FUNCTION_BLOCK FB_Evt_EventClasses EXTENDS FB_BA_View
VAR
	{region 'Standard'}
		// Intention:				Demonstration of a standard use-case:
		//							- Declaration of event classes for desired event-types and alarm-modes.
		//							  (See "FB_BA_EC01" for complete example of this standard use-case).
		//							- Applies event behaviour that just works.
		EC_Std01					: FB_BA_EC := (
										iParent							:= THIS^,
										nInstanceID						:= 200,
										sDescription					:= '{Standard EC (Extended Alarm)}',
										eEventType						:= E_BA_EventType.eAlarm,
										eAlarmMode						:= E_BA_AlarmMode.eExtended
									);
		EC_Std02					: FB_BA_EC := (
										iParent							:= THIS^,
										nInstanceID						:= 201,
										sDescription					:= '{Standard EC (Standard Alarm)}',
										eEventType						:= E_BA_EventType.eAlarm,
										eAlarmMode						:= E_BA_AlarmMode.eStandard
									);
		EC_Std03					: FB_BA_EC := (
										iParent							:= THIS^,
										nInstanceID						:= 202,
										sDescription					:= '{Standard EC (Simple Alarm)}',
										eEventType						:= E_BA_EventType.eAlarm,
										eAlarmMode						:= E_BA_AlarmMode.eSimple
									);

		// Intention:				Assignment of an object's event class reference.
		SimpleAlm01					: FB_BA_BI := (
										iParent							:= THIS^,
										sDescription					:= '{Some simple alarm}',
										nEventClassID					:= 202,
										sInactiveText					:= 'Normal',
										sActiveText						:= 'Alarm'
									);
	{endregion}
	{region 'Customize default settings'}
		// Intention:				Demonstration of customizing events default behaviour by settings modification:
		//							- No difference in code to "standard use-case".
		//							  (Use implementation of the same event classes)
		//							- The following parameters are editable per alarm-mode (See "BA_Param"):
		//							  - Acknowledge Flags
		//							  - Event Enable Flags
		
		// Sample:					How to adjust the default-settings of event-classes?
		//							- No acknowledgement should be required for any "simple" events.
		//							  BA_Param.aAckFlags_Simple := [ FALSE, FALSE, FALSE ];
	{endregion}
	{region 'Individual parameters'}
		// Intention:				Demonstration of customizing individual event-classes and objects:
		// 							- Initialization of an event-classes "AcknowledgeRequired" flags.
		EC_Cstm01					: FB_BA_EC := (
										iParent							:= THIS^,
										nInstanceID						:= 220,
										sDescription					:= '{Customized EC (Alarm 1)}',
										eEventType						:= E_BA_EventType.eAlarm,
										aAcknowledgeRequired			:= [ TRUE, TRUE, TRUE ]
									);
		EC_Cstm02					: FB_BA_EC := (
										iParent							:= THIS^,
										nInstanceID						:= 221,
										sDescription					:= '{Customized EC (Alarm 2)}',
										eEventType						:= E_BA_EventType.eAlarm,
										aAcknowledgeRequired			:= [ TRUE, FALSE, FALSE ]
									);
		EC_Cstm03					: FB_BA_EC := (
										iParent							:= THIS^,
										nInstanceID						:= 222,
										sDescription					:= '{Customized EC (Alarm 3)}',
										eEventType						:= E_BA_EventType.eAlarm,
										aAcknowledgeRequired			:= [ FALSE, FALSE, FALSE ]
									);
										 
		// Sample:					How to initialize individual objects?
		// Intention:				- Assignment of an object's event class reference.
		// 							- Initialization of an object's "EventEnable" flags.
		Alm01						: FB_BA_BI := (
										iParent							:= THIS^,
										sDescription					:= '{Some alarm without acknowledgement}',
										nEventClassID					:= 222,
										aEventEnable					:= [ TRUE, TRUE, TRUE ],
										sInactiveText					:= 'Normal',
										sActiveText						:= 'Alarm'
									);
		Alm02						: FB_BA_BI := (
										iParent							:= THIS^,
										sDescription					:= '{Some alarm with acknowledgement}',
										nEventClassID					:= 220,
										aEventEnable					:= [ TRUE, TRUE, TRUE ],
										sInactiveText					:= 'Normal',
										sActiveText						:= 'Alarm'
									);
	{endregion}
END_VAR

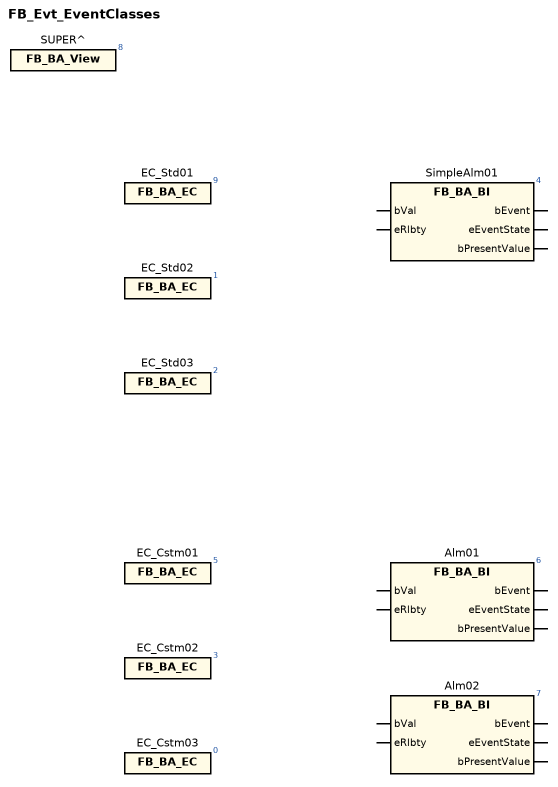
EC_Cstm03(); // FB_BA_EC
EC_Std02(); // FB_BA_EC
EC_Std03(); // FB_BA_EC
EC_Cstm02(); // FB_BA_EC
SimpleAlm01(); // FB_BA_BI
EC_Cstm01(); // FB_BA_EC
Alm01(); // FB_BA_BI
Alm02(); // FB_BA_BI
SUPER^(); // FB_BA_View
EC_Std01(); // FB_BA_EC

END_FUNCTION_BLOCK

(* stored: Version 1.1.0.1, ProductVersion 3.1.4024.9
   POU FB_Evt_EventClasses: Id {0ca2e0b8-0ddb-4496-9651-2def95d8dec6}, SpecialFunc None *)
